// SIMATIC S7-200 project (STEP 7-Micro/WIN), CPU 222 REL 02.01

SYMBOL_TABLE USUARIO1
MARCHA           I0.0
LAMPARA          Q0.0
END_SYMBOL_TABLE

ORGANIZATION_BLOCK PRINCIPAL:OB1
TITLE=COMENTARIOS DEL PROGRAMA
BEGIN
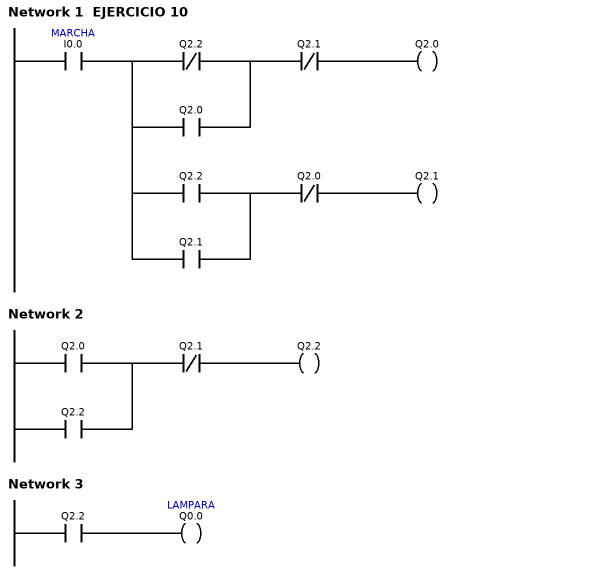
Network 1 // EJERCICIO 10
LD     MARCHA:I0.0
LPS
LDN    Q2.2
O      Q2.0
ALD
AN     Q2.1
=      Q2.0
LPP
LD     Q2.2
O      Q2.1
ALD
AN     Q2.0
=      Q2.1
Network 2
LD     Q2.0
O      Q2.2
AN     Q2.1
=      Q2.2
Network 3
LD     Q2.2
=      LAMPARA:Q0.0
END_ORGANIZATION_BLOCK
